{attribute 'GeneratedUsingTerminal: EK1122-0000-0018'}
{attribute addProperty BoxType "EK1122-0000-0018"}
{attribute addProperty Id "Beckhoff_ER3xxxsub_EK1100EK1100_1FC0878B2A_0001_ER3174_0002_0016ER3174_DCC7866252A_0002_ER3174_0002_0022ER3174_DCC7866252A_0003_ER3174_0002_0023ER3174_DCC7866252A_0004_ER3184_0002_0019ER3184_DCC7866252A_0005_ER3184_0002_0020ER3184_DCC7866252A_0006_ER3184_0002_0021ER3184_DCC7866252A_0007_ER3184_1002_0020ER3184_DCC7866252A_0008_ER3184_1002_0021ER3184_DCC7866252A_0009_ER3204_0002_0016ER3204_6CD7E11952A_0010_ER3204_0002_0020ER3204_6CD7E11952A_0011_ER3204_0002_0021ER3204_AB25C3AC48A_0012_ER3314_0002_0021ER3314_E65CDB1C48"}
{attribute addProperty CRC "1334719193"}
{attribute addProperty Size "618"}
{attribute addProperty Name "Beckhoff ER3xxxEK1122"}
TYPE Beckhoff_ER3xxxEK1122_4F8E32D9 EXTENDS EK1122_1FC0878B :
STRUCT
	{attribute addProperty Name "Beckhoff ER3xxxsub EK1100"}
	{attribute addProperty PreviousPort "Beckhoff ER3xxxEK1122 : D"}
	Beckhoff_ER3xxxsub_EK1100 : EK1100_1FC0878B;
	{attribute addProperty Name "A_0001(ER3174-0002-0016)"}
	{attribute addProperty PreviousPort "Beckhoff ER3xxxsub EK1100 : C"}
	A_0001_ER3174_0002_0016 : ER3174_DCC78662;
	{attribute addProperty Name "A_0002(ER3174-0002-0022)"}
	{attribute addProperty PreviousPort "A_0001(ER3174-0002-0016) : B"}
	A_0002_ER3174_0002_0022 : ER3174_DCC78662;
	{attribute addProperty Name "A_0003(ER3174-0002-0023)"}
	{attribute addProperty PreviousPort "A_0002(ER3174-0002-0022) : B"}
	A_0003_ER3174_0002_0023 : ER3174_DCC78662;
	{attribute addProperty Name "A_0004(ER3184-0002-0019)"}
	{attribute addProperty PreviousPort "A_0003(ER3174-0002-0023) : B"}
	A_0004_ER3184_0002_0019 : ER3184_DCC78662;
	{attribute addProperty Name "A_0005(ER3184-0002-0020)"}
	{attribute addProperty PreviousPort "A_0004(ER3184-0002-0019) : B"}
	A_0005_ER3184_0002_0020 : ER3184_DCC78662;
	{attribute addProperty Name "A_0006(ER3184-0002-0021)"}
	{attribute addProperty PreviousPort "A_0005(ER3184-0002-0020) : B"}
	A_0006_ER3184_0002_0021 : ER3184_DCC78662;
	{attribute addProperty Name "A_0007(ER3184-1002-0020)"}
	{attribute addProperty PreviousPort "A_0006(ER3184-0002-0021) : B"}
	A_0007_ER3184_1002_0020 : ER3184_DCC78662;
	{attribute addProperty Name "A_0008(ER3184-1002-0021)"}
	{attribute addProperty PreviousPort "A_0007(ER3184-1002-0020) : B"}
	A_0008_ER3184_1002_0021 : ER3184_DCC78662;
	{attribute addProperty Name "A_0009(ER3204-0002-0016)"}
	{attribute addProperty PreviousPort "A_0008(ER3184-1002-0021) : B"}
	A_0009_ER3204_0002_0016 : ER3204_6CD7E119;
	{attribute addProperty Name "A_0010(ER3204-0002-0020)"}
	{attribute addProperty PreviousPort "A_0009(ER3204-0002-0016) : B"}
	A_0010_ER3204_0002_0020 : ER3204_6CD7E119;
	{attribute addProperty Name "A_0011(ER3204-0002-0021)"}
	{attribute addProperty PreviousPort "A_0010(ER3204-0002-0020) : B"}
	A_0011_ER3204_0002_0021 : ER3204_AB25C3AC;
	{attribute addProperty Name "A_0012(ER3314-0002-0021)"}
	{attribute addProperty PreviousPort "A_0011(ER3204-0002-0021) : B"}
	A_0012_ER3314_0002_0021 : ER3314_E65CDB1C;
END_STRUCT
END_TYPE

(* stored: Version 1.2.0.0, ProductVersion 3.1.4024.11
   DUT Beckhoff_ER3xxxEK1122_4F8E32D9: Id {e5fd0e2a-2e29-4420-a4cd-77ae72f0ecb6} *)
